//{attribute 'qualified_only'}
VAR_GLOBAL
	GAB_FactoryIO_Inputs : ARRAY [0..1] OF WORD;
	GAB_FactoryIO_InputRegs : ARRAY [0..7] OF INT;
	GAB_FactoryIO_Outputs : ARRAY [0..1] OF WORD;
	GAB_FactoryIO_OutputsRegs : ARRAY [0..7] OF INT;
END_VAR

(* stored: Version 1.1.0.1, ProductVersion 3.1.4024.11
   GVL GVL_FactoryIO: Id {a4883462-1cb0-43b2-bb87-d6ce56b75e06} *)
